{attribute 'qualified_only'}
{attribute 'strict'}
{attribute 'to_string'}
TYPE E_Command :
(
	Forward := 0,
	Stop := 1,
	Backward := 2,
	Generate := 3
);
END_TYPE

(* stored: Version 1.1.0.1, ProductVersion 3.1.4024.12
   DUT E_Command: Id {8d37bf0a-9f06-498f-993f-692835782342} *)
